Universal Robots PolyScope program: Ching_Field_2_SDR.urp

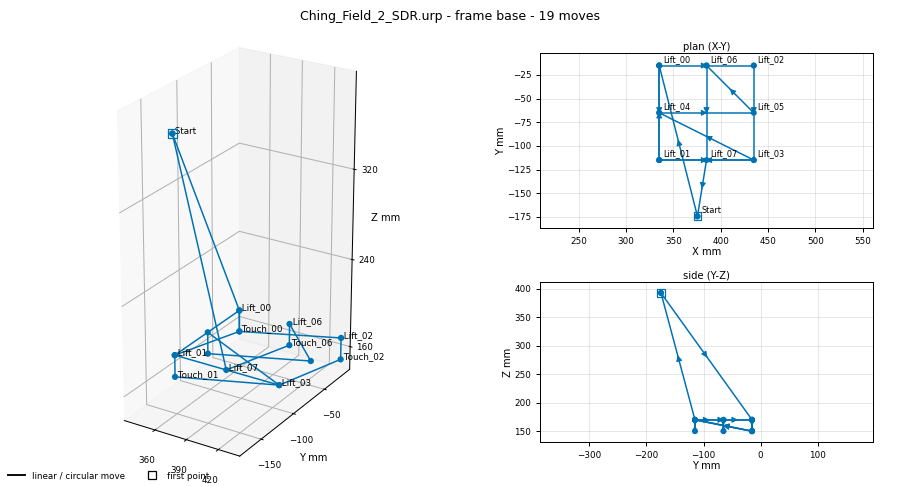
[picture p0: tool path of Ching_Field_2_SDR.urp in frame base, 19 of 19 moves have a stored position in this frame; points joined in program order, loops and branches not executed]
Program Ching_Field_2_SDR (installation=default directory=/programs createdIn=5.11.5.1010327 lastSavedIn=5.11.9.1010452 robotSerialNumber=20225200364)
Calibrated DH parameters: a=[0.00002, -0.569483, -0.54992, -0.00001, -0.000036, 0]; d=[0.180894, -146.691669, 192.918669, -46.053088, 0.119778, 0.115602]; alpha=[1.571425, -0.001534, 0.003359, 1.568739, -1.571477, 0]; deltaTheta=[0, 0.376258, -0.101074, -0.275185, -0.000002, 0]
Robot Program (runOnlyOnce=false)
  MoveL speed 150 mm/s, acceleration 1200 mm/s^2 (useActiveTCP=true) feature=Base
    Waypoint Start: TCP in base x=375.438 y=-174.524 z=392.25 mm, rx=2.2167 ry=2.2232 rz=-0.002 rad; joints [-0.006, -90.002, -120.024, -239.98, -90.047, 0.072] deg; TCP offset x=0 y=0 z=0 mm, rx=0 ry=0 rz=0 rad
    Waypoint Lift_00: TCP in base x=335 y=-15 z=170 mm, rx=2.221 ry=2.221 rz=0 rad; joints [28.81, -101.437, -138.766, -209.826, -90.082, 29.149] deg; TCP offset x=0 y=0 z=0 mm, rx=0 ry=0 rz=0 rad
    Waypoint Touch_00: motionParameters(jointSpeed=1.047198 jointAcceleration=1.396263 cartesianSpeed=0.005 cartesianAcceleration=1.2); TCP in base x=335 y=-15 z=150 mm, rx=2.221 ry=2.221 rz=0 rad; joints [28.812, -103.943, -139.239, -206.847, -90.071, 29.159] deg; TCP offset x=0 y=0 z=0 mm, rx=0 ry=0 rz=0 rad
      Until TOOL_CONTACT_DETECTION (allowActions=false retraction=-0.0003 decelerationAcceleration=3 decelerationAngularAcceleration=34.906585)
    MoveDirectionNode (selectedDirection=YMinus) feature=Base
      Until DISTANCE (allowActions=false deceleration=3 distanceNodeType=STOP) Distance=0.1; motionParameters(blendRadius=0)
    Waypoint Lift_01: TCP in base x=335 y=-115 z=170 mm, rx=2.221 ry=2.221 rz=0 rad; joints [10.577, -102.96, -136.551, -210.507, -90.086, 10.915] deg; TCP offset x=0 y=0 z=0 mm, rx=0 ry=0 rz=0 rad
    Waypoint Lift_00: TCP in base x=335 y=-15 z=170 mm, rx=2.221 ry=2.221 rz=0 rad; joints [28.81, -101.437, -138.766, -209.826, -90.082, 29.149] deg; TCP offset x=0 y=0 z=0 mm, rx=0 ry=0 rz=0 rad
    Waypoint Touch_00: motionParameters(jointSpeed=1.047198 jointAcceleration=1.396263 cartesianSpeed=0.005 cartesianAcceleration=1.2); TCP in base x=335 y=-15 z=150 mm, rx=2.221 ry=2.221 rz=0 rad; joints [28.812, -103.943, -139.239, -206.847, -90.071, 29.159] deg; TCP offset x=0 y=0 z=0 mm, rx=0 ry=0 rz=0 rad
      Until TOOL_CONTACT_DETECTION (allowActions=false retraction=-0.0003 decelerationAcceleration=3 decelerationAngularAcceleration=34.906585)
    MoveDirectionNode (selectedDirection=XPlus) feature=Base
      Until DISTANCE (allowActions=false deceleration=3 distanceNodeType=STOP) Distance=0.1; motionParameters(blendRadius=0)
    Waypoint Lift_02: TCP in base x=435 y=-15 z=170 mm, rx=2.221 ry=2.221 rz=0 rad; joints [21.646, -109.024, -127.128, -213.873, -90.081, 21.976] deg; TCP offset x=0 y=0 z=0 mm, rx=0 ry=0 rz=0 rad
    Waypoint Touch_02: motionParameters(jointSpeed=1.047198 jointAcceleration=1.396263 cartesianSpeed=0.005 cartesianAcceleration=1.2); TCP in base x=435 y=-15 z=150 mm, rx=2.221 ry=2.221 rz=0 rad; joints [21.647, -111.002, -127.518, -211.505, -90.073, 21.983] deg; TCP offset x=0 y=0 z=0 mm, rx=0 ry=0 rz=0 rad
      Until TOOL_CONTACT_DETECTION (allowActions=false retraction=-0.0003 decelerationAcceleration=3 decelerationAngularAcceleration=34.906585)
    MoveDirectionNode (selectedDirection=YMinus) feature=Base
      Until DISTANCE (allowActions=false deceleration=3 distanceNodeType=STOP) Distance=0.1; motionParameters(blendRadius=0)
    Waypoint Lift_03: TCP in base x=435 y=-115 z=170 mm, rx=2.221 ry=2.221 rz=0 rad; joints [7.993, -110.065, -125.42, -214.532, -90.085, 8.321] deg; TCP offset x=0 y=0 z=0 mm, rx=0 ry=0 rz=0 rad
    Waypoint Lift_01: TCP in base x=335 y=-115 z=170 mm, rx=2.221 ry=2.221 rz=0 rad; joints [10.577, -102.96, -136.551, -210.507, -90.086, 10.915] deg; TCP offset x=0 y=0 z=0 mm, rx=0 ry=0 rz=0 rad
    Waypoint Touch_01: motionParameters(jointSpeed=1.047198 jointAcceleration=1.396263 cartesianSpeed=0.005 cartesianAcceleration=1.2); TCP in base x=335 y=-115 z=150 mm, rx=2.221 ry=2.221 rz=0 rad; joints [10.579, -105.344, -137.004, -207.671, -90.076, 10.924] deg; TCP offset x=0 y=0 z=0 mm, rx=0 ry=0 rz=0 rad
      Until TOOL_CONTACT_DETECTION (allowActions=false retraction=-0.0003 decelerationAcceleration=3 decelerationAngularAcceleration=34.906585)
    MoveDirectionNode (selectedDirection=XPlus) feature=Base
      Until DISTANCE (allowActions=false deceleration=3 distanceNodeType=STOP) Distance=0.1; motionParameters(blendRadius=0)
    Waypoint Lift_03: TCP in base x=435 y=-115 z=170 mm, rx=2.221 ry=2.221 rz=0 rad; joints [7.993, -110.065, -125.42, -214.532, -90.085, 8.321] deg; TCP offset x=0 y=0 z=0 mm, rx=0 ry=0 rz=0 rad
    Waypoint Lift_04: TCP in base x=335 y=-65 z=170 mm, rx=2.221 ry=2.221 rz=0 rad; joints [19.787, -101.921, -138.07, -210.033, -90.084, 20.126] deg; TCP offset x=0 y=0 z=0 mm, rx=0 ry=0 rz=0 rad
    Waypoint Touch_04: motionParameters(jointSpeed=1.047198 jointAcceleration=1.396263 cartesianSpeed=0.005 cartesianAcceleration=1.2); TCP in base x=335 y=-65 z=150 mm, rx=2.221 ry=2.221 rz=0 rad; joints [19.789, -104.386, -138.536, -207.101, -90.073, 20.135] deg; TCP offset x=0 y=0 z=0 mm, rx=0 ry=0 rz=0 rad
      Until TOOL_CONTACT_DETECTION (allowActions=false retraction=-0.0003 decelerationAcceleration=3 decelerationAngularAcceleration=34.906585)
    MoveDirectionNode (selectedDirection=XPlus) feature=Base
      Until DISTANCE (allowActions=false deceleration=3 distanceNodeType=STOP) Distance=0.1; motionParameters(blendRadius=0)
    Waypoint Lift_05: TCP in base x=435 y=-65 z=170 mm, rx=2.221 ry=2.221 rz=0 rad; joints [14.861, -109.349, -126.597, -214.075, -90.083, 15.19] deg; TCP offset x=0 y=0 z=0 mm, rx=0 ry=0 rz=0 rad
    Waypoint Lift_06: TCP in base x=385 y=-15 z=170 mm, rx=2.221 ry=2.221 rz=0 rad; joints [24.697, -105.367, -132.926, -211.733, -90.081, 25.033] deg; TCP offset x=0 y=0 z=0 mm, rx=0 ry=0 rz=0 rad
    Waypoint Touch_06: motionParameters(jointSpeed=1.047198 jointAcceleration=1.396263 cartesianSpeed=0.005 cartesianAcceleration=1.2); TCP in base x=385 y=-15 z=150 mm, rx=2.221 ry=2.221 rz=0 rad; joints [24.699, -107.574, -133.351, -209.101, -90.072, 25.041] deg; TCP offset x=0 y=0 z=0 mm, rx=0 ry=0 rz=0 rad
      Until TOOL_CONTACT_DETECTION (allowActions=false retraction=-0.0003 decelerationAcceleration=3 decelerationAngularAcceleration=34.906585)
    MoveDirectionNode (selectedDirection=YMinus)
      Until DISTANCE (allowActions=false deceleration=3 distanceNodeType=STOP) Distance=0.1; motionParameters(blendRadius=0)
    Waypoint Lift_07: TCP in base x=385 y=-115 z=170 mm, rx=2.221 ry=2.221 rz=0 rad; joints [9.101, -106.596, -131.01, -212.412, -90.086, 9.435] deg; TCP offset x=0 y=0 z=0 mm, rx=0 ry=0 rz=0 rad
    Waypoint Start: TCP in base x=375.438 y=-174.524 z=392.25 mm, rx=2.2167 ry=2.2232 rz=-0.002 rad; joints [-0.006, -90.002, -120.024, -239.98, -90.047, 0.072] deg; TCP offset x=0 y=0 z=0 mm, rx=0 ry=0 rz=0 rad
    Halt
